ABB RAPID module: Left_ASL_Demo.mod

MODULE Left_ASL_Demo
LOCAL CONST string YuMi_App_Program_Version:="1.0.1"; !Do not edit or remove this line!
LOCAL VAR robtarget s60 := [[519.08,52.62,111.62],[0.0190745,-0.317014,0.947041,-0.0474542],[-2,1,-2,11],[179.331,9E+09,9E+09,9E+09,9E+09,9E+09]];
LOCAL VAR robtarget s59 := [[430.39,123.37,180.80],[0.0999607,0.310832,0.943756,0.0521077],[-2,1,0,11],[131.707,9E+09,9E+09,9E+09,9E+09,9E+09]];
LOCAL VAR robtarget s58 := [[358.29,68.30,132.84],[0.2751,-0.0426083,0.86319,-0.421199],[-1,1,0,11],[117.327,9E+09,9E+09,9E+09,9E+09,9E+09]];
LOCAL VAR robtarget s57 := [[358.29,68.30,132.84],[0.275101,-0.0426095,0.86319,-0.421198],[-1,1,0,11],[117.327,9E+09,9E+09,9E+09,9E+09,9E+09]];
LOCAL VAR robtarget s56 := [[488.88,196.13,-9.51],[0.0436672,0.774832,-0.594672,-0.209984],[-2,0,-2,11],[-128.122,9E+09,9E+09,9E+09,9E+09,9E+09]];
LOCAL VAR robtarget s55 := [[438.93,-11.04,-14.27],[0.137086,0.640295,-0.744056,-0.132704],[-2,0,-2,11],[-135.659,9E+09,9E+09,9E+09,9E+09,9E+09]];
LOCAL VAR robtarget s54 := [[346.07,2.52,-21.90],[0.183409,0.628509,-0.722146,-0.223252],[-2,0,-2,11],[-129.96,9E+09,9E+09,9E+09,9E+09,9E+09]];
LOCAL VAR robtarget s53 := [[346.07,2.53,-21.91],[0.183395,0.628507,-0.722154,-0.223247],[-2,0,-2,11],[-129.96,9E+09,9E+09,9E+09,9E+09,9E+09]];
LOCAL VAR robtarget s52 := [[346.36,2.76,-22.07],[0.182499,0.628074,-0.72283,-0.223011],[-2,0,-2,11],[-129.954,9E+09,9E+09,9E+09,9E+09,9E+09]];
LOCAL VAR robtarget s51 := [[346.36,2.76,-22.07],[0.182498,0.628074,-0.722831,-0.22301],[-2,0,-2,11],[-129.954,9E+09,9E+09,9E+09,9E+09,9E+09]];
LOCAL VAR robtarget s50 := [[346.36,2.76,-22.07],[0.182497,0.628073,-0.722832,-0.223009],[-2,0,-2,11],[-129.954,9E+09,9E+09,9E+09,9E+09,9E+09]];
LOCAL VAR robtarget s49 := [[346.36,2.76,-22.07],[0.182493,0.628073,-0.722833,-0.22301],[-2,0,-2,11],[-129.954,9E+09,9E+09,9E+09,9E+09,9E+09]];
LOCAL VAR robtarget s48 := [[346.36,2.76,-22.07],[0.182492,0.628071,-0.722834,-0.223011],[-2,0,-2,11],[-129.954,9E+09,9E+09,9E+09,9E+09,9E+09]];
LOCAL VAR robtarget s47 := [[346.36,2.76,-22.07],[0.182489,0.628071,-0.722835,-0.22301],[-2,0,-2,11],[-129.954,9E+09,9E+09,9E+09,9E+09,9E+09]];
LOCAL VAR robtarget s46 := [[346.37,2.77,-22.07],[0.182481,0.628066,-0.722841,-0.223011],[-2,0,-2,11],[-129.954,9E+09,9E+09,9E+09,9E+09,9E+09]];
LOCAL VAR robtarget s45 := [[346.37,2.77,-22.08],[0.182475,0.628061,-0.722847,-0.22301],[-2,0,-2,11],[-129.954,9E+09,9E+09,9E+09,9E+09,9E+09]];
LOCAL VAR robtarget s44 := [[346.37,2.77,-22.08],[0.182471,0.628058,-0.722852,-0.223008],[-2,0,-2,11],[-129.954,9E+09,9E+09,9E+09,9E+09,9E+09]];
LOCAL VAR robtarget s43 := [[346.37,2.77,-22.08],[0.182457,0.628053,-0.72286,-0.223006],[-2,0,-2,11],[-129.954,9E+09,9E+09,9E+09,9E+09,9E+09]];
LOCAL VAR robtarget s42 := [[346.39,2.81,-22.09],[0.182382,0.628009,-0.722913,-0.223019],[-2,0,-2,11],[-129.952,9E+09,9E+09,9E+09,9E+09,9E+09]];
LOCAL VAR robtarget s41 := [[346.92,3.05,-22.39],[0.18104,0.627419,-0.724003,-0.222238],[-2,0,-2,11],[-129.95,9E+09,9E+09,9E+09,9E+09,9E+09]];
LOCAL VAR robtarget s40 := [[367.84,3.92,14.47],[0.223286,0.640903,-0.702206,-0.215161],[-2,0,-2,11],[-130.827,9E+09,9E+09,9E+09,9E+09,9E+09]];
LOCAL VAR robtarget s39 := [[412.30,51.52,46.99],[0.26981,0.654674,-0.703812,-0.0570357],[-2,0,-2,11],[-126.803,9E+09,9E+09,9E+09,9E+09,9E+09]];
LOCAL VAR robtarget s38 := [[496.94,50.54,-0.50],[0.0852698,-0.611194,0.718186,-0.321526],[-2,0,-1,1010],[-139.426,9E+09,9E+09,9E+09,9E+09,9E+09]];
LOCAL VAR robtarget s37 := [[500.11,217.09,68.79],[0.372259,-0.540285,0.603529,-0.453064],[-2,0,-1,1010],[-136.231,9E+09,9E+09,9E+09,9E+09,9E+09]];
LOCAL VAR robtarget s36 := [[409.25,103.49,24.74],[0.422813,-0.52314,0.597648,-0.436314],[-2,0,-1,1010],[-146.03,9E+09,9E+09,9E+09,9E+09,9E+09]];
LOCAL VAR robtarget s35 := [[321.14,2.68,-3.70],[0.326511,-0.570175,0.616333,-0.434079],[-2,0,-1,1010],[-149.503,9E+09,9E+09,9E+09,9E+09,9E+09]];
LOCAL VAR robtarget s34 := [[323.71,20.37,-12.88],[0.347699,-0.567053,0.614733,-0.423862],[-2,0,-1,1010],[-149.327,9E+09,9E+09,9E+09,9E+09,9E+09]];
LOCAL VAR robtarget s33 := [[318.83,3.47,-66.12],[0.377646,-0.544178,0.635778,-0.396283],[-2,0,-1,1010],[-148.179,9E+09,9E+09,9E+09,9E+09,9E+09]];
LOCAL VAR robtarget s32 := [[319.84,5.22,-58.84],[0.383222,-0.546134,0.616372,-0.418288],[-2,0,-1,1010],[-147.982,9E+09,9E+09,9E+09,9E+09,9E+09]];
LOCAL VAR robtarget s31 := [[328.17,3.84,-35.32],[0.291971,-0.584613,0.689413,-0.312553],[-2,0,-1,1010],[-148.669,9E+09,9E+09,9E+09,9E+09,9E+09]];
LOCAL VAR robtarget s30 := [[337.64,30.76,-7.64],[0.0603166,-0.700953,0.706625,-0.0755479],[-2,-1,-1,1010],[-140.725,9E+09,9E+09,9E+09,9E+09,9E+09]];
LOCAL VAR robtarget s29 := [[332.62,43.68,-12.15],[0.0965366,0.657321,-0.744356,0.0674054],[-2,-1,-1,1010],[-139.929,9E+09,9E+09,9E+09,9E+09,9E+09]];
LOCAL VAR robtarget s28 := [[357.26,47.13,-18.41],[0.0647535,-0.627827,0.773446,-0.0585039],[-2,-1,-1,1010],[-144.37,9E+09,9E+09,9E+09,9E+09,9E+09]];
LOCAL VAR robtarget s27 := [[280.93,-22.19,-89.26],[0.280661,0.753652,-0.552241,-0.219698],[-2,-2,0,1010],[-144.058,9E+09,9E+09,9E+09,9E+09,9E+09]];
LOCAL VAR robtarget s26 := [[411.50,234.48,-12.30],[0.0247232,-0.893074,-0.44509,-0.0608532],[-2,1,0,11],[-112.468,9E+09,9E+09,9E+09,9E+09,9E+09]];
LOCAL VAR robtarget s25 := [[452.81,0.61,-28.01],[0.0534624,-0.733061,-0.678059,0.000726626],[-2,1,0,11],[-120.866,9E+09,9E+09,9E+09,9E+09,9E+09]];
LOCAL VAR robtarget s24 := [[349.20,3.29,-30.65],[0.132352,-0.755431,-0.636905,0.0784733],[-2,0,0,11],[-116.649,9E+09,9E+09,9E+09,9E+09,9E+09]];
LOCAL VAR robtarget s23 := [[349.20,3.30,-30.65],[0.132356,-0.755432,-0.636904,0.0784701],[-2,0,0,11],[-116.649,9E+09,9E+09,9E+09,9E+09,9E+09]];
LOCAL VAR robtarget s22 := [[349.20,3.30,-30.65],[0.132359,-0.75544,-0.636895,0.0784554],[-2,0,0,11],[-116.649,9E+09,9E+09,9E+09,9E+09,9E+09]];
LOCAL VAR robtarget s21 := [[350.41,3.36,-31.57],[0.13288,-0.758459,-0.633307,0.0774998],[-2,0,0,11],[-116.715,9E+09,9E+09,9E+09,9E+09,9E+09]];
LOCAL VAR robtarget s20 := [[350.41,3.35,-31.57],[0.132858,-0.758463,-0.633305,0.0775062],[-2,0,0,11],[-116.715,9E+09,9E+09,9E+09,9E+09,9E+09]];
LOCAL VAR robtarget s19 := [[350.73,4.94,-30.75],[0.143302,-0.746172,-0.646652,0.0673269],[-2,0,0,11],[-116.784,9E+09,9E+09,9E+09,9E+09,9E+09]];
LOCAL VAR robtarget s18 := [[350.73,4.94,-30.75],[0.143304,-0.746172,-0.646652,0.0673253],[-2,0,0,11],[-116.784,9E+09,9E+09,9E+09,9E+09,9E+09]];
LOCAL VAR robtarget s17 := [[350.78,4.97,-30.77],[0.143293,-0.746154,-0.646681,0.0672732],[-2,0,0,11],[-116.784,9E+09,9E+09,9E+09,9E+09,9E+09]];
LOCAL VAR robtarget s16 := [[350.78,4.97,-30.77],[0.143296,-0.746154,-0.64668,0.0672737],[-2,0,0,11],[-116.783,9E+09,9E+09,9E+09,9E+09,9E+09]];
LOCAL VAR robtarget s15 := [[352.15,0.79,-30.13],[0.123754,-0.784046,-0.604348,0.0687036],[-2,1,0,11],[-116.948,9E+09,9E+09,9E+09,9E+09,9E+09]];
LOCAL VAR robtarget s14 := [[352.14,0.80,-30.14],[0.123767,-0.784023,-0.604376,0.0687027],[-2,1,0,11],[-116.946,9E+09,9E+09,9E+09,9E+09,9E+09]];
LOCAL VAR robtarget s13 := [[371.04,-4.26,-8.95],[0.102659,-0.801009,-0.587171,0.0554594],[-2,1,0,11],[-118.371,9E+09,9E+09,9E+09,9E+09,9E+09]];
LOCAL VAR robtarget s12 := [[489.39,-45.07,-15.89],[0.201984,0.597068,0.764634,-0.13434],[-2,1,-1,11],[-123.487,9E+09,9E+09,9E+09,9E+09,9E+09]];
LOCAL VAR robtarget s11 := [[532.50,100.52,35.86],[0.416487,-0.209336,0.789097,-0.400052],[-2,0,-1,1010],[-145.784,9E+09,9E+09,9E+09,9E+09,9E+09]];
LOCAL VAR robtarget s10 := [[319.95,-0.66,-0.80],[0.308284,-0.570712,0.646516,-0.40158],[-2,0,-1,1010],[-145.404,9E+09,9E+09,9E+09,9E+09,9E+09]];
LOCAL VAR robtarget s9 := [[317.46,2.30,-64.05],[0.377499,-0.534834,0.655031,-0.377334],[-2,0,-1,1010],[-151.879,9E+09,9E+09,9E+09,9E+09,9E+09]];
LOCAL VAR robtarget s8 := [[319.86,0.63,-56.51],[0.390843,-0.522879,0.647092,-0.393842],[-2,0,-1,1010],[-151.437,9E+09,9E+09,9E+09,9E+09,9E+09]];
LOCAL VAR robtarget s7 := [[357.76,22.39,-2.64],[0.0696524,-0.606296,0.775248,-0.162923],[-2,-1,-1,1010],[-145.265,9E+09,9E+09,9E+09,9E+09,9E+09]];
LOCAL VAR robtarget s6 := [[339.22,39.97,2.31],[0.254333,0.704549,-0.624556,-0.221031],[-2,-2,0,1010],[-142.847,9E+09,9E+09,9E+09,9E+09,9E+09]];
LOCAL VAR robtarget s5 := [[282.32,-20.83,-89.42],[0.275747,0.742915,-0.569862,-0.217482],[-2,-2,0,1010],[-144.216,9E+09,9E+09,9E+09,9E+09,9E+09]];
LOCAL VAR robtarget s4 := [[292.39,7.25,-43.65],[0.06839,0.68191,-0.727285,0.0371075],[-2,-1,-1,1010],[-144.963,9E+09,9E+09,9E+09,9E+09,9E+09]];
LOCAL VAR robtarget s3 := [[286.48,-20.76,-86.12],[0.126721,0.794038,-0.590704,-0.0671829],[-2,-1,-1,1010],[-143.981,9E+09,9E+09,9E+09,9E+09,9E+09]];
LOCAL VAR robtarget s2 := [[304.13,-11.50,-50.26],[0.0519145,0.826957,-0.559517,-0.0197134],[-2,-1,-1,1010],[-154.754,9E+09,9E+09,9E+09,9E+09,9E+09]];
LOCAL VAR robtarget s1 := [[316.65,45.52,21.47],[0.0502929,0.702983,-0.635561,0.315196],[-1,0,-1,1010],[-169.577,9E+09,9E+09,9E+09,9E+09,9E+09]];
PROC main()
MoveSync s57;
OpenHand;
MoveSync s1;
MoveSync s2;
MoveSync s3;
MoveSync s5;
MoveSync s27;
CloseHand;
MoveSync s6;
MoveSync s30;
MoveSync s31;
MoveSync s32;
MoveSync s33;
OpenHand;
MoveSync s34;
MoveSync s35;
MoveSync s36;
MoveSync s37;
MoveSync s38;
MoveSync s39;
MoveSync s40;
MoveSync s41;
CloseHand;
MoveSync s42;
MoveSync s43;
MoveSync s44;
MoveSync s45;
MoveSync s46;
MoveSync s47;
MoveSync s48;
MoveSync s49;
MoveSync s50;
MoveSync s51;
MoveSync s52;
MoveSync s54;
OpenHand;
MoveSync s55;
MoveSync s56;
MoveSync s60;
MoveSync s58;
ENDPROC
ENDMODULE
